FUNCTION_BLOCK FB_TILT_TEST
VAR_INPUT
END_VAR
VAR_OUTPUT
END_VAR
VAR
END_VAR

END_FUNCTION_BLOCK

(* stored: Version 1.1.0.1, ProductVersion 3.1.4024.12
   POU FB_TILT_TEST: Id {fb59190b-17af-4192-a83b-6e0804f23142}, SpecialFunc None *)
